FUNCTION_BLOCK FB_HydraulicsMain
VAR CONSTANT
	sCycleStateTextDef: ARRAY[0..20]  OF STRING :=	
		['State 0: Wait for Start',
		'State 1: Check Oil temperature and oil levels and Check all valves are in de-energised state',
		'State 2: When pump is running start the cooler and filterpump',
		'State 3: When pumps are running open circulation valve',
		'State 4: Check ciruclation valve is open, open Accumlator valve',
		'State 5: Check if Accu valve is open, and wait 15s',
		'State 6: Open the blocking valve',
		'State 7: Check if the blocking valve is open, and if pressure > x',
		'State 8: Main Hydraulics running',
		'State 9: Check if all analog valves are in the safe state',
		'State 10: Close presurize pumpvalve, stop cooling fan and filtermotor',
		'State 11: Close blocking valve and stop pump',
		'State 12: Spare',
		'State 13: [Paused: Close blocking valve]',
		'State 14: [Paused: Awaiting Restart]',
		'State 15: [Stopped Direct]'];
	
	tCycleStateTimeouts: ARRAY[0..10] OF TIME := 
		[T#10S,T#10S,T#10S,T#10S,T#10S,T#10S,T#10S,T#10S,T#10S,T#10S,
		T#10S];

	sInitStateTextDef: ARRAY[0..10] OF STRING :=
		['State 0: Wait for Init Start',
		'State 1: Await pressure relief',
		'State 2: Move up',
		'State 3: Description Init State 3',
		'State 4: Description Init State 4',
		'State 5: Description Init State 5',
		'State 6: Description Init State 6',
		'State 7: Description Init State 7',
		'State 8: Description Init State 8',
		'State 9: Description Init State 9',
		'State 10: Stop init state'];

	tInitStateTimeouts: ARRAY[0..10] OF TIME := 
		[T#10S,T#10S,T#10S,T#10S,T#10S,T#10S,T#10S,T#10S,T#10S,T#10S
		,T#10S];
END_VAR
VAR_INPUT
	mxReset								: BOOL;	(*Reset Error*)
	mxEmergency							: BOOL; // Used when a emergency stop button was pushed.
	mxDoorOpened						: BOOL;	// Used when a door was opened in the system
	mxAutoMode							: BOOL; (* TRUE = Automode *)
	PlcCycleTime						: REAL;
	
	
	
	(*State vars*)
	mxResetCycleState					: BOOL;
	mxResetInitState					: BOOL;
END_VAR
VAR_IN_OUT
	MachineParameters					: ST_HydraulicsMainMachPar;
END_VAR
VAR_OUTPUT
(*Errors*)
	Errors								: ST_HydraulicsMainErrors;
	mxErrorInit							: BOOL;		(* Error, stop immediately. Initialisation neccesary *)
	mxErrorStopinPos					: BOOL;		(* Error, stop in position. Only reset neccesary *)
	
	(* State vars *)
	mxCycleBusy							: BOOL;
	mxInitbusy							: BOOL;
	mxCycleInPause						: BOOL;
(* Vars *)
	mxInitialized						: BOOL;
	
	mxHydraulicsReady					: BOOL;
END_VAR
VAR
	(* State vars *)
	miCycleState					: INT :=0;
	miCycleOldstate					: INT :=0;
	mxCycleTransitionState			: BOOL := FALSE;
	sCycleStateText					: STRING;
	exCycleTimeOut					: BOOL;		(* Timeout for the whole programcycle *)
	CycleTimeout					: TON;
	CycleTimeOutUpFlank				: R_TRIG;
	mxCycleTimeoutEnable			: BOOL;
	CycleTime						: REAL;
	mxCycleHasError					: BOOL;
	miStopState						: INT;
	mxStartCycle					: BOOL;
	mxStopCycle						: BOOL;
	mxStopDirect					: BOOL;
	mxStopCycleEmpty				: BOOL;
	
	miInitState						: INT	:=0;
	miInitOldstate					: INT	:=0;
	mxInitTransitionState			: BOOL	:= FALSE;
	sInitStateText					: STRING;
	exInitTimeOut					: BOOL;		(* Timeout for the whole programcycle *)
	InitTimeout						: TON;
	InitTimeOutUpFlank				: R_TRIG;
	mxInitTimeoutEnable				: BOOL;
	InitTime						: REAL;
	mxInitHasError					: BOOL;
	mxStartInit						: BOOL;
	mxStopInit						: BOOL;	

	ixHydraulicsMcc24vError				AT %I*: BOOL;
	ixCabinetCoolerError				At %I*: BOOL;
	
	ixTemperatureSwitch40c				AT %I*: BOOL;
	ixTemperatureSwitch55c				AT %I*: BOOL;
	ixTemperatureSwitchTooHigh			AT %I*: BOOL;
	
	ixPressureFilterAt75				AT %I*: BOOL;
	ixPressureFilterAt100				AT %I*: BOOL;
	
	ixAuxFilterAt75						AT %I*: BOOL;
	ixAuxFilterAt100					AT %I*: BOOL;
	
	ixOilLvlTooLow						AT %I*: BOOL;
	ixOilLvlLow							AT %I*: BOOL;
	
	FT_AutoMode							: F_TRIG;
	
	(* Objects *)
	HydraulicPump						: FB_MotorSS;
	FilterMotor							: FB_Motor;
	CoolingFan							: FB_Motor;
	
	PressurizePumpValve					: FB_MonoValveNoFdbck;
	AccuDrainValve						: FB_MonoValveNoFdbck;
	IsolationValve						: FB_MonoValveNoFdbck;
	
	OilTemperature						: FB_AnalogIn4_20mA;
	MainSystemPressure					: FB_AnalogIn4_20mA;
	
	HmiForceCool						: BOOL;
	FT_ForceCool						: F_TRIG;
	T_DelayOpenBlockingValve			: TON;
	SR_TempTooHigh						: SR;
	SR_LevelTooLow						: SR;
	SR_Filter100Dirty					: SR;
	SR_AuxFilter100Dirty				: SR;
	SR_Filter75DirtyWarning				: SR;
	SR_AuxFilter75DirtyWarning			: SR;

	SR_CabinetCoolerError				: SR;
	SR_HydraulicsMcc24VError			: SR;
	RT_Doorsopenend						: R_TRIG;	// Used to produce a situation that is safe when doors are openend, but is also quick in restarting the machine
	
	mxTest1								: BOOL;
	T_DepresurizePump					: TON;
	RT_OilCoolerOn						: R_TRIG;
	FT_OilCoolerOff						: F_TRIG;
	FT_Emergency						: F_Trig;
	
	mxTest5: BOOL;
	RT_EmergencyStop: R_TRIG;

	T_CheckFeedback: TON;
END_VAR

Cycle();
Error();
Objects();

// If both emergencies become zero, recheck if cooler needs to run.
FT_Emergency(CLK:=mxEmergency OR mxDoorOpened);
RT_OilCoolerOn(CLK:=ixTemperatureSwitch55c);
FT_OilCoolerOff (CLK:=ixTemperatureSwitch40c);

IF ((RT_OilCoolerOn.q) OR (FT_Emergency.Q AND ixTemperatureSwitch55c)) AND NOT CoolingFan.IsRunning THEN
	CoolingFan.M_Start();
END_IF

IF FT_OilCoolerOff.q AND CoolingFan.IsRunning THEN
	CoolingFan.M_Stop();
END_IF

METHOD M_StartCycle : BOOL
IF NOT mxCycleBusy OR mxCycleInPause THEN
	mxStartCycle:= TRUE;	
	mxStopCycle:=False;
END_IF
END_METHOD

ACTION Objects:
OilTemperature(
	EngLowLimit:= -25, 
	EngUpperLimit:= 100); (* In °C *)

PressurizePumpValve(
	mxReset:= mxReset, 
	mxEmergency:=mxEmergency , 
	mxAutoMode:=mxAutoMode , 
	RHSR_Blocked:= , 
	SlowValveIsInverted:= , 
	mxDisableManualAutoTrigger:=TRUE,
	mxIsOn=> );
	
	
	// special situation, on door opened keep the accu drain valve openend.
AccuDrainValve(
	mxReset:= mxReset, 
	mxEmergency:= mxDoorOpened, 
	mxAutoMode:=mxAutoMode , 
	RHSR_Blocked:= , 
	SlowValveIsInverted:= , 
	mxDisableManualAutoTrigger:=TRUE,
	mxIsOn=> );
	
IsolationValve(
	mxReset:= mxReset, 
	mxEmergency:=mxEmergency , 
	mxAutoMode:=mxAutoMode , 
	RHSR_Blocked:= , 
	SlowValveIsInverted:= , 
	mxDisableManualAutoTrigger:=TRUE,
	mxIsOn=> );
	
HydraulicPump(
	mxReset:= mxReset, 
	mxEmergency:= mxEmergency,
	mxAutoMode:= mxAutoMode,
	mxDisableManualAutoTrigger:=TRUE,
	Errors=> Errors.HydraulicPump);
	
FilterMotor(
	mxReset:= mxReset, 
	mxEmergency:= mxEmergency, 
	mxAutoMode:= mxAutoMode, 
	mxDisableManualAutoTrigger:=TRUE,
	Errors=>Errors.FilterMotor);
	
CoolingFan(
	mxReset:= mxReset, 
	mxEmergency:= mxEmergency,
	mxAutoMode:= mxAutoMode,
	mxDisableManualAutoTrigger:=TRUE,
	Errors=> Errors.Coolingfan);
	
MainSystemPressure(
	EngLowLimit:=0, 
	EngUpperLimit:=315, 
	maOut=> , 
	EngUnits=> , 
	EngFilt=> , 
	OverRange=> , 
	UnderRange=> );
END_ACTION

METHOD M_StopInit
;
END_METHOD

METHOD M_StopCycle : BOOL
IF mxCycleBusy THEN 
	mxStopCycle:= TRUE; 
END_IF
END_METHOD

METHOD M_StopDirect

IF mxCycleBusy THEN
	mxStopDirect:= TRUE;	
END_IF
END_METHOD

ACTION Cycle:
(*StateChange (Transition)  Signalgeneration*)
mxCycleTransitionState:=(miCycleState<>miCycleOldstate);
(*State text*)
sCycleStateText:=sCycleStateTextDef[miCycleState];
(*Timeout Watchdog for Statemachine*)
mxCycleTimeoutEnable:=NOT (miCycleState=0) AND NOT mxReset;

CycleTimeout(IN:=mxCycleTimeoutEnable  , PT:=tCycleStateTimeouts[miCycleState] );
CycleTimeOutUpFlank(CLK:=CycleTimeout.Q );
miCycleOldstate:=miCycleState;

(*Set Errorbit when Raising edge of Timeout has been detected*)
IF CycleTimeOutUpFlank.Q THEN
	exCycleTimeOut:=TRUE; 			(* 1 Timeout for the whole programcycle *)
END_IF

(*Function to reset the Statemachine*)
IF mxResetCycleState THEN
	mxResetCycleState:= FALSE;
	mxInitialized := FALSE;
		
	miCycleState:=0;
	mxCycleTransitionState:=FALSE;

	mxStartCycle:= FALSE;
	mxStopCycle:= FALSE;
	mxStopDirect:=FALSE;
	mxStopcycleEmpty:=False;
	
	HydraulicPump.M_Stop();
	CoolingFan.M_Stop();
	FilterMotor.M_Stop();
	AccuDrainValve.M_Off();
	IsolationValve.M_Off();
	PressurizePumpValve.M_Off();
END_IF

mxCycleHasError:=FALSE;

T_DelayOpenBlockingValve(PT:= T#15S);
T_DepresurizePump(PT:=T#2S);
T_CheckFeedback(PT:=T#300MS);

mxHydraulicsReady:= miCycleState=8;


(*Cycle State's*)
CASE miCycleState OF

	0:	// Idle state/Wait for start
		IF mxStopDirect THEN
			mxStopDirect:= FALSE;		
			miCycleState:= 15;
		ELSIF mxStopCycle THEN		
			miCycleState:= 0;
			mxStopCycle:=FALSE;
		ELSIF mxStartCycle THEN		
			miCycleState:= 1;
			mxStartCycle:=FALSE;
			mxStopCycleEmpty:=FALSE;
		END_IF	

	1:	// Check oil temperature and oil levels	and valves Start main pump
		IF mxStopDirect THEN
			mxStopDirect:= FALSE;
			miCycleState:= 15;
		ELSIF mxStopCycle THEN
			mxStopCycle:= FALSE;
			miStopState:= miCycleState;
			miCycleState:= 13;
		ELSIF ixTemperatureSwitchTooHigh AND ixOilLvlTooLow AND NOT PressurizePumpValve.mxIsOn THEN			
			HydraulicPump.M_Start();
			miCycleState:= 2;
		END_IF

	2:	//When pump is running, start cooler and filterpump 	
		IF mxStopDirect THEN
			mxStopDirect:= FALSE;
			miCycleState:= 15;
		ELSIF mxStopCycle THEN
			mxStopCycle:= FALSE;
			miStopState:= miCycleState;
			miCycleState:= 13;
		ELSIF HydraulicPump.IsRunning THEN			
			FilterMotor.M_Start();
			miCycleState:= 3;
		END_IF

	3:	//When pumps are running open the Pressurize valve 
		IF mxStopDirect THEN
			mxStopDirect:= FALSE;			
			miCycleState:= 15;
		ELSIF mxStopCycle THEN
			mxStopCycle:= FALSE;
			miStopState:= miCycleState;
			miCycleState:= 13;
		ELSIF FilterMotor.IsRunning THEN					
			PressurizePumpValve.M_On();
			miCycleState:= 4;
		END_IF
	
	4:	// (P) When circulation valve is open, open accumulator valve
		IF mxStopDirect THEN
			mxStopDirect:= FALSE;		
			miCycleState:= 15;
		ELSIF mxStopCycle THEN
			mxStopCycle:= FALSE;
			miStopState:= miCycleState;
			miCycleState:= 13;
		ELSIF PressurizePumpValve.mxIsOn THEN			
			AccuDrainValve.M_On();
			miCycleState:= 5;
		END_IF
	
	5:	// (P) Check if accuValve is open and wait for 15s 
		IF mxStopDirect THEN
			mxStopDirect:= FALSE;		
			miCycleState:= 15;
		ELSIF mxStopCycle THEN
			mxStopCycle:= FALSE;
			miStopState:= miCycleState;
			miCycleState:= 13;
		ELSIF AccuDrainValve.mxIsOn THEN			
			T_DelayOpenBlockingValve.IN:=TRUE;
			miCycleState:= 6;
		END_IF
		
	6:	// (NP) Open blocking valve
		IF mxStopDirect THEN
			mxStopDirect:= FALSE;	
			miCycleState:= 15;
		ELSIF T_DelayOpenBlockingValve.Q THEN				
			T_DelayOpenBlockingValve.IN:=FALSE;
			IsolationValve.M_On();
			miCycleState:= 7;
		END_IF
		
	7:	// (NP) Check if blocking valve is open and main pressure is > X 
		IF mxStopDirect THEN
			mxStopDirect:= FALSE;
			miCycleState:= 15;
		ELSIF IsolationValve.mxIsOn AND (MainSystemPressure.EngFilt > 240.0) THEN			
			miCycleState:= 8;
		END_IF
		
	8: // State of main hydraulics is running, wait in this step for stop.	
		IF mxStopDirect THEN
			mxStopDirect:= FALSE;
			miCycleState:= 15;
		ELSIF mxStopCycle THEN				// To pause
			mxStopCycle:= FALSE;
			miStopState:= miCycleState;
			miCycleState:= 13;
		ELSIF mxStopCycleEmpty THEN 		// Stopping the cycle CMD.
			mxStopCycleEmpty:=FALSE;
			miStopState:= miCycleState;
			miCycleState:= 9;
		END_IF
		
	9:	// Check if all analog valves are in safe state. (not controlled)
		IF mxStopDirect THEN
			mxStopDirect:= FALSE;
			miCycleState:= 15;
		ELSIF mxStopCycle THEN		
			mxStopCycle:= FALSE;
			miStopState:= miCycleState;
			miCycleState:= 13;
		ELSIF (MAIN.InMoldDrying.TopMoldA.HydraulicCilinder.SafePosReached AND 
			Main.InMoldDrying.TopMoldB.HydraulicCilinder.SafePosReached AND 
			Main.InMoldDrying.TransferMold.HydraulicCilinder.SafePosReached) THEN
			PressurizePumpValve.M_Off();	// Pomp vrijschakelen
			CoolingFan.M_Stop();
			FilterMotor.M_Stop();
			
			T_DepresurizePump.IN := TRUE;
			
			miCycleState:=10;
		END_IF
		
	10:	// Check if pressurise pump valve, coolingfan / filtermotor are stopped/closed -> Open isolation and drain valve
		IF mxStopDirect THEN
			mxStopDirect:= FALSE;
			miCycleState:= 15;
		ELSIF mxStopCycle THEN		
			mxStopCycle:= FALSE;
			miStopState:= miCycleState;
			miCycleState:= 13;
		ELSIF NOT PressurizePumpValve.mxIsOn AND NOT CoolingFan.IsRunning AND NOT FilterMotor.IsRunning AND T_DepresurizePump.Q THEN
			T_DepresurizePump.IN := FALSE;	
			IsolationValve.M_Off();
			AccuDrainValve.M_Off();
			micycleState:=11;
		END_IF
		
	11:	// Check if isolationvalve and accudrain valve have stopped -> stop pump
		IF mxStopDirect THEN
			mxStopDirect:= FALSE;
			miCycleState:= 15;
		ELSIF mxStopCycle THEN		
			mxStopCycle:= FALSE;
			miStopState:= miCycleState;
			miCycleState:= 13;
		ELSIF NOT IsolationValve.mxIsOn AND NOT AccuDrainValve.mxIsOn THEN	
			HydraulicPump.M_Stop();
			miCycleState:=0;
		END_IF
		
	13:	// [Pause cycle] Close blocking valve
		IF mxStopDirect THEN
			mxStopDirect:= FALSE;
			miCycleState:= 15;
		ELSE
 			IsolationValve.M_Off();		// Switch off the isolation valve in rest mode (rest of hydraulics keep functioning as normal).
			T_CheckFeedback.In :=TRUE;	
			miCycleState:=14;					
		END_IF
		
	14: // [Paused] cycle step.			
		IF mxStopDirect OR (T_CheckFeedback.q AND (MAIN.Errors.InMoldDryingErrors.TopMoldA.Hydraulic.SafePositionValveNotReached OR
		Main.Errors.InMoldDryingErrors.TopMoldB.Hydraulic.SafePositionValveNotReached OR
		Main.Errors.InMoldDryingErrors.TransferMold.HydraulicCilinder.SafePositionValveNotReached)) THEN
			T_CheckFeedback.In :=FALSE;
			mxStopDirect:= FALSE;
			miCycleState:= 15;
		ELSIF mxStartCycle THEN
			mxStopCycle:=FALSE;
			mxStartCycle:=FALSE;
			T_CheckFeedback.In :=FALSE;
 			IsolationValve.M_on();		// At restart, open valve again.
			miCycleState:=miStopState;
		ELSIF mxStopCycleEmpty THEN		// At pause stop rest of hydraulics.
			mxStopcycleEmpty:=FALSE;
			T_CheckFeedback.In :=FALSE;
			miCycleState := 9;
		END_IF

	15:	// Stop Direct
		mxStartCycle:= FALSE;
		mxStopCycle:= FALSE;
		mxStopCycleEmpty:=FALSE;
		mxInitialized:= FALSE;
		
		HydraulicPump.M_Stop();
		CoolingFan.M_Stop();
		FilterMotor.M_Stop();
		
		IsolationValve.M_Off();
		PressurizePumpValve.M_Off();
		AccuDrainValve.M_Off();		
		
		miCycleState:= 0;
END_CASE

mxCycleBusy:= miCycleState<>0;
mxCycleInPause := miCycleState=14;
END_ACTION

METHOD M_StopCycleEmpty : BOOL
IF mxCycleBusy THEN 
	mxStopCycleEmpty:= TRUE; 
END_IF
END_METHOD

ACTION Error:

SR_TempTooHigh(SET1:=NOT ixTemperatureSwitchTooHigh, RESET:=mxReset , Q1=>Errors.OilTemperatureTooHigh);
SR_LevelTooLow(SET1:=NOT ixOilLvlTooLow, Reset:=mxReset, Q1=>Errors.OilLevelTooLow);

SR_Filter100Dirty(SET1:=NOT ixPressureFilterAt100, RESET:=mxReset, Q1=>Errors.Filter100Dirty);
SR_AuxFilter100Dirty(SET1:=NOT ixAuxFilterAt100, RESET:=mxReset, Q1=>Errors.AuxFilter100Dirty);

SR_Filter75DirtyWarning(SET1:=ixPressureFilterAt75, RESET:=mxReset, Q1=>Errors.Filter75Dirty);
SR_AuxFilter75DirtyWarning(SET1:=ixAuxFilterAt75, RESET:=mxReset, Q1=>Errors.AuxFilter75Dirty);

SR_CabinetCoolerError(SET1:= NOT ixCabinetCoolerError, Reset:=mxReset, Q1=>);

SR_HydraulicsMcc24VError(SET1:= NOT ixHydraulicsMcc24vError, Reset:=mxReset, Q1=>);


RT_Doorsopenend(CLK:=mxDoorOpened);
RT_EmergencyStop(CLK:=mxEmergency);

IF RT_Doorsopenend.Q THEN
	M_StopCycle();
END_IF

IF RT_EmergencyStop.Q THEN
	M_StopDirect();
END_IF



(**********************************************************************************************************)
mxErrorStopinPos:=  FALSE;

mxErrorInit:= HydraulicPump.mxErrorInit OR Errors.Filter100Dirty OR Errors.AuxFilter100Dirty OR Errors.OilLevelTooLow OR
				Errors.OilTemperatureTooHigh OR FilterMotor.mxErrorInit OR CoolingFan.mxErrorInit;
END_ACTION

END_FUNCTION_BLOCK

(* stored: Version 1.1.0.1, ProductVersion 3.1.4020.12
   POU FB_HydraulicsMain: Id {3981de64-156d-4ad8-80a2-78d705ffb77f}, SpecialFunc None
   Method M_StartCycle: Id {23c82821-bb4b-42f7-b56a-4ec9995d96cf}
   Action Objects: Id {63170b63-f4cd-4429-ac1b-df5e730ad407}
   Method M_StopInit: Id {70b250cf-0b9a-4fa7-93bb-6dc13ce4e146}
   Method M_StopCycle: Id {7bf68905-085e-4b1f-81f6-4006fb1101d3}
   Method M_StopDirect: Id {9e8558f0-e4fa-4bb7-8256-f18c40d3f5ef}
   Action Cycle: Id {c3cff216-476b-49a2-8b2f-6e28d426d6e6}
   Method M_StopCycleEmpty: Id {e3cc7dc4-d945-4e94-adea-d2238685669b}
   Action Error: Id {fdad504a-67ea-46f2-be61-4d24b55ec8c0} *)
